// TwinCAT 3 PLC project Vaten
// ProgramVersion: 3.1.4024.0
// libraries:
//   Tc2_Standard, * (Beckhoff Automation GmbH)
//   Tc2_System, * (Beckhoff Automation GmbH)
//   Tc3_Module, * (Beckhoff Automation GmbH)
// project tree:
//   / GlobalTextList.TcGTLO, PlcTask.TcTTO, Visualization Manager.TcVMO (not stored)
//   POUs/ MAIN.TcPOU
//   VISUs/ Visualization.TcVIS
// (motion and I/O tree: see PLC project potentiometer_inlezen)
// real-time tasks:
//   TASK PlcTask: cycle T#10ms, priority 20, ADS port 350
//   TASK PlcTask1: cycle T#10ms, priority 21, ADS port 351
//   TASK PlcTask2: cycle T#10ms, priority 22, ADS port 352
//   TASK PlcTask3: cycle T#10ms, priority 26, ADS port 353
//   TASK PlcTask4: cycle T#10ms, priority 25, ADS port 354
//   TASK PlcTask5: cycle T#10ms, priority 24, ADS port 355
//   TASK PlcTask6: cycle T#10ms, priority 23, ADS port 356
//   TASK PlcTask7: cycle T#10ms, priority 27, ADS port 357

CONFIGURATION Vaten
    RESOURCE PLC ON TwinCAT3
        TASK PlcTask(INTERVAL := T#10ms, PRIORITY := 27);
        PROGRAM MAIN WITH PlcTask : MAIN;
    END_RESOURCE
END_CONFIGURATION

// ---- POUs/MAIN.TcPOU
PROGRAM MAIN
VAR
// Analoge ingangen
	nSensor1              AT %I*:LREAL;
	nSensor2              AT %I*:LREAL;
	nSensor3              AT %I*:LREAL;
	
// Analoge uitgangen
	nVat1                 AT %Q*:LREAL;//MAX2000L
    nVat2                 AT %Q*:LREAL;//MAX3000L
	nVat3                 AT %Q*:LREAL;//MAX5000L
	nBardisplay           AT %Q*:LREAL;
	
END_VAR

(*
Vaten

De inhoud van 3 vaten wordt afzonderlijk gemeten en kunnen maximaal 2000L, 3000L en 5000L bevatten. 
De waarde die men inleest is de hoeveelheid die zich in het vat bevindt (nVat1, nVat2 en nVat3). 

Simuleer deze ingangen. 
Bouw een visualisatie die de inhoud van elke tank afzonderlijk alsook de som weergeeft. 
Maak gebruik van 3 sliders en 1 bar display. Houd eveneens rekening met de maximum waarden.
*)

// BELANGRIJK:
// Controleer de instellingen/verschalingen bij de visualisatie voor een beter begrip

nVat1:=100.0*(nSensor1/2000.0);
nVat2:=100.0*(nSensor2/3000.0);
nVat3:=100.0*(nSensor3/5000.0);
nBardisplay:=nVat1+nVat2+nVat3;

END_PROGRAM

// ---- GlobalTextList.TcGTLO
TEXTLIST GlobalTextList
  10 = 'Sensor1'
  634 = 'Sensor2'
  535 = 'Sensor3'
  937 = 'Som van de vaten'
  764 = 'Vat1'
  14 = 'Vat2'
  236 = 'Vat3'
END_TEXTLIST

// ---- VISUs/Visualization.TcVIS
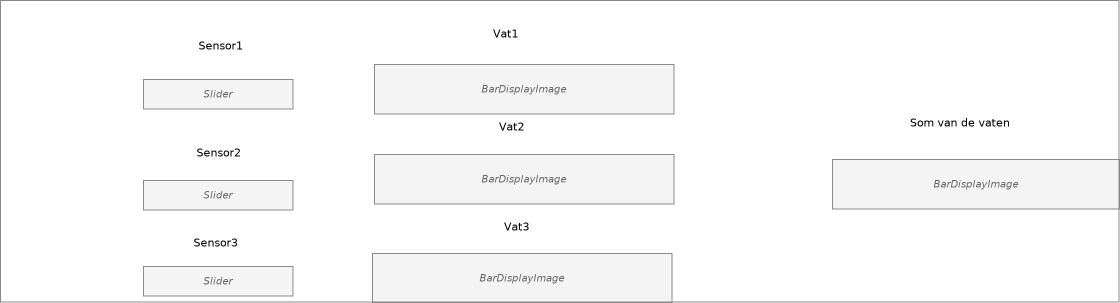
VISUALIZATION Visualization  // 1120x303
    Slider (143,79 150x30), variable: MAIN.nSensor1, scale 0..2000
    Slider (143,180 150x30), variable: MAIN.nSensor2, scale 0..3000
    Slider (143,266 150x30), variable: MAIN.nSensor3, scale 0..5000
    BarDisplayImage (374,64 300x50), value: MAIN.nVat1, style: BarDisplayImage-Gray, scale format: %.1f, scale 0..100
    BarDisplayImage (832,159 288x50), value: MAIN.nBardisplay, style: BarDisplayImage-Gray, scale format: %.1f, scale 0..300
    BarDisplayImage (374,154 300x50), value: MAIN.nVat2, style: BarDisplayImage-Gray, scale format: %.1f, scale 0..100
    BarDisplayImage (372,253 300x50), value: MAIN.nVat3, style: BarDisplayImage-Gray, scale format: %.1f, scale 0..100
    Label (146,31 150x30), "Sensor1"
    Label (144,138 150x30), "Sensor2"
    Label (141,228 150x30), "Sensor3"
    Label (431,19 150x30), "Vat1"
    Label (437,112 150x30), "Vat2"
    Label (442,212 150x30), "Vat3"
    Label (885,108 150x30), "Som van de vaten"
END_VISUALIZATION
